{attribute 'TcGenerated'}
{attribute 'no-analysis'}
{attribute 'linkalways'}
// This function has been automatically generated from the project information.
VAR_GLOBAL CONSTANT
	{attribute 'const_non_replaced'}
	stLibVersion_CNM_AssertionInterfaceTests : ST_LibVersion := (iMajor := 1, iMinor := 2, iBuild := 0, iRevision := 6, nFlags := 0, sVersion := '1.2.0.6');
END_VAR

(* stored: Version 1.1.0.1, ProductVersion 3.1.4026.13
   GVL Global_Version: Id {653167b4-b317-49a7-aceb-644c5f3907d2} *)
